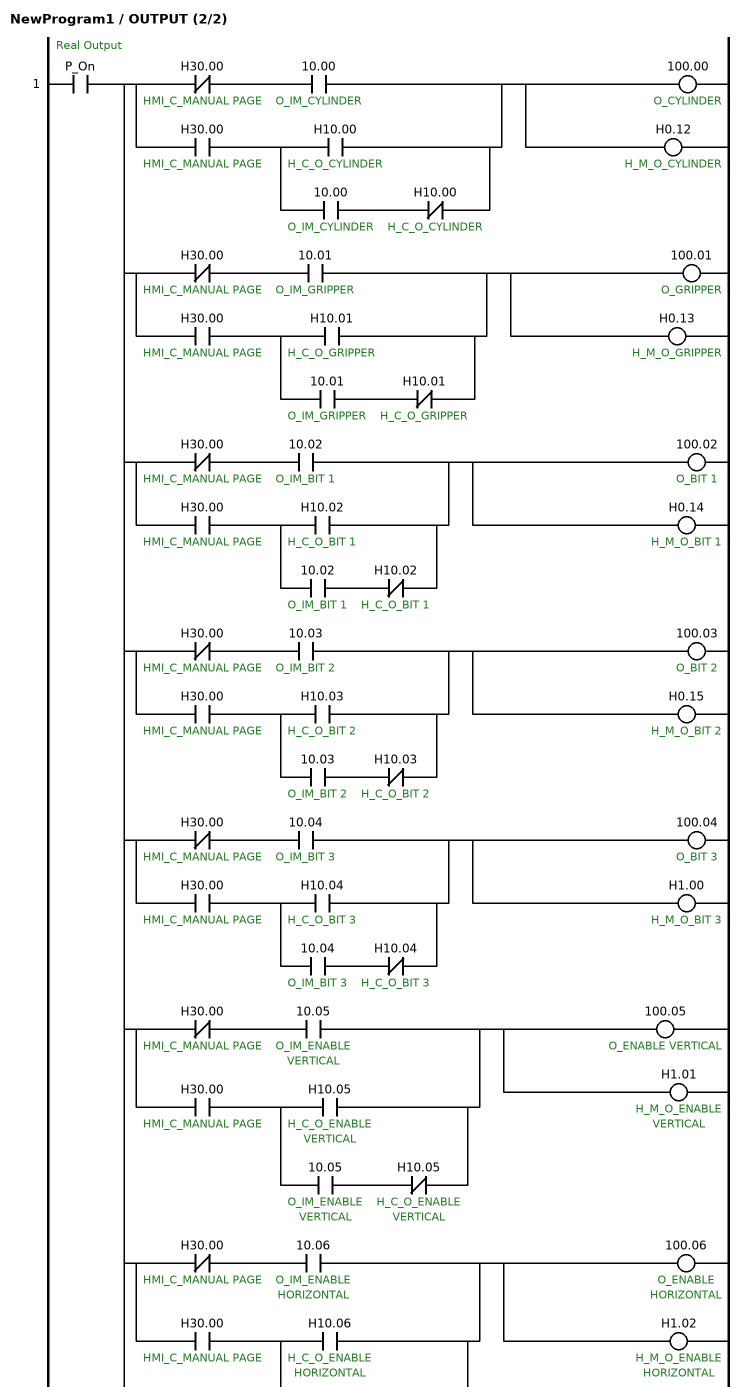
; [picture p48: NewProgram1 / OUTPUT, rungs 1-1]

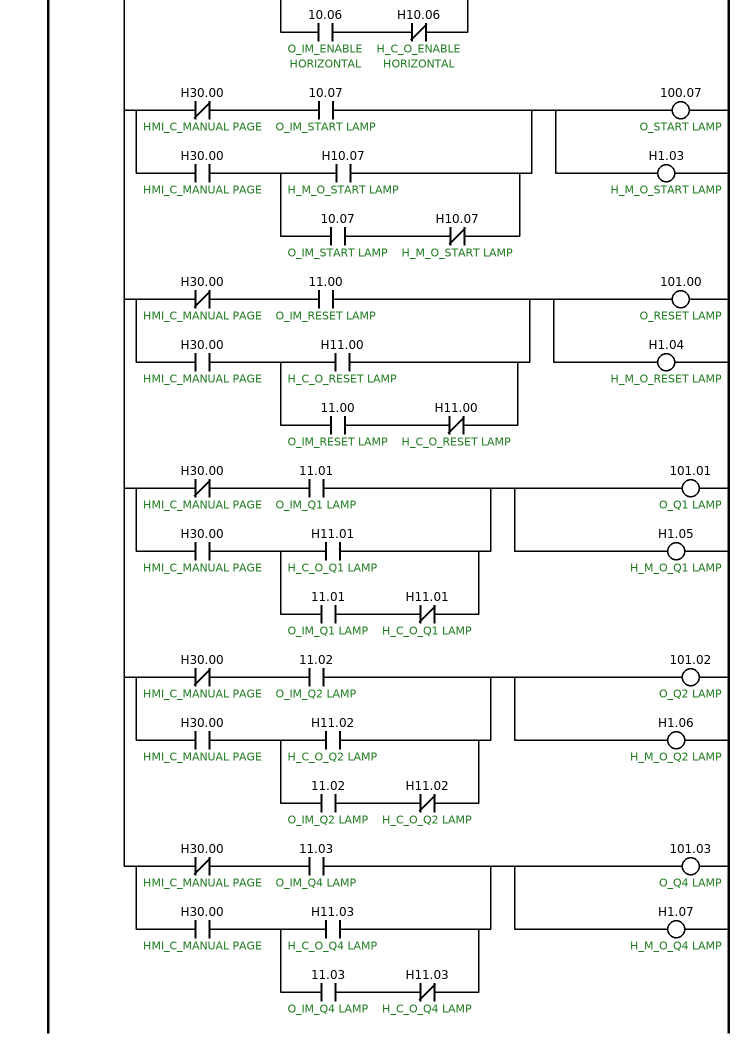
; rung 1: Real Output
LD P_On
OUT TR0
LDNOT H30.00  ; HMI_C_MANUAL PAGE
AND 10.00  ; O_IM_CYLINDER
LD H30.00  ; HMI_C_MANUAL PAGE
LD H10.00  ; H_C_O_CYLINDER
LD 10.00  ; O_IM_CYLINDER
ANDNOT H10.00  ; H_C_O_CYLINDER
ORLD
ANDLD
ORLD
ANDLD
OUT 100.00  ; O_CYLINDER
OUT H0.12  ; H_M_O_CYLINDER
LD TR0
LDNOT H30.00  ; HMI_C_MANUAL PAGE
AND 10.01  ; O_IM_GRIPPER
LD H30.00  ; HMI_C_MANUAL PAGE
LD H10.01  ; H_C_O_GRIPPER
LD 10.01  ; O_IM_GRIPPER
ANDNOT H10.01  ; H_C_O_GRIPPER
ORLD
ANDLD
ORLD
ANDLD
OUT 100.01  ; O_GRIPPER
OUT H0.13  ; H_M_O_GRIPPER
LD TR0
LDNOT H30.00  ; HMI_C_MANUAL PAGE
AND 10.02  ; O_IM_BIT 1
LD H30.00  ; HMI_C_MANUAL PAGE
LD H10.02  ; H_C_O_BIT 1
LD 10.02  ; O_IM_BIT 1
ANDNOT H10.02  ; H_C_O_BIT 1
ORLD
ANDLD
ORLD
ANDLD
OUT 100.02  ; O_BIT 1
OUT H0.14  ; H_M_O_BIT 1
LD TR0
LDNOT H30.00  ; HMI_C_MANUAL PAGE
AND 10.03  ; O_IM_BIT 2
LD H30.00  ; HMI_C_MANUAL PAGE
LD H10.03  ; H_C_O_BIT 2
LD 10.03  ; O_IM_BIT 2
ANDNOT H10.03  ; H_C_O_BIT 2
ORLD
ANDLD
ORLD
ANDLD
OUT 100.03  ; O_BIT 2
OUT H0.15  ; H_M_O_BIT 2
LD TR0
LDNOT H30.00  ; HMI_C_MANUAL PAGE
AND 10.04  ; O_IM_BIT 3
LD H30.00  ; HMI_C_MANUAL PAGE
LD H10.04  ; H_C_O_BIT 3
LD 10.04  ; O_IM_BIT 3
ANDNOT H10.04  ; H_C_O_BIT 3
ORLD
ANDLD
ORLD
ANDLD
OUT 100.04  ; O_BIT 3
OUT H1.00  ; H_M_O_BIT 3
LD TR0
LDNOT H30.00  ; HMI_C_MANUAL PAGE
AND 10.05  ; O_IM_ENABLE VERTICAL
LD H30.00  ; HMI_C_MANUAL PAGE
LD H10.05  ; H_C_O_ENABLE VERTICAL
LD 10.05  ; O_IM_ENABLE VERTICAL
ANDNOT H10.05  ; H_C_O_ENABLE VERTICAL
ORLD
ANDLD
ORLD
ANDLD
OUT 100.05  ; O_ENABLE VERTICAL
OUT H1.01  ; H_M_O_ENABLE VERTICAL
LD TR0
LDNOT H30.00  ; HMI_C_MANUAL PAGE
AND 10.06  ; O_IM_ENABLE HORIZONTAL
LD H30.00  ; HMI_C_MANUAL PAGE
LD H10.06  ; H_C_O_ENABLE HORIZONTAL
LD 10.06  ; O_IM_ENABLE HORIZONTAL
ANDNOT H10.06  ; H_C_O_ENABLE HORIZONTAL
ORLD
ANDLD
ORLD
ANDLD
OUT 100.06  ; O_ENABLE HORIZONTAL
OUT H1.02  ; H_M_O_ENABLE HORIZONTAL
LD TR0
LDNOT H30.00  ; HMI_C_MANUAL PAGE
AND 10.07  ; O_IM_START LAMP
LD H30.00  ; HMI_C_MANUAL PAGE
LD H10.07  ; H_M_O_START LAMP
LD 10.07  ; O_IM_START LAMP
ANDNOT H10.07  ; H_M_O_START LAMP
ORLD
ANDLD
ORLD
ANDLD
OUT 100.07  ; O_START LAMP
OUT H1.03  ; H_M_O_START LAMP
LD TR0
LDNOT H30.00  ; HMI_C_MANUAL PAGE
AND 11.00  ; O_IM_RESET LAMP
LD H30.00  ; HMI_C_MANUAL PAGE
LD H11.00  ; H_C_O_RESET LAMP
LD 11.00  ; O_IM_RESET LAMP
ANDNOT H11.00  ; H_C_O_RESET LAMP
ORLD
ANDLD
ORLD
ANDLD
OUT 101.00  ; O_RESET LAMP
OUT H1.04  ; H_M_O_RESET LAMP
LD TR0
LDNOT H30.00  ; HMI_C_MANUAL PAGE
AND 11.01  ; O_IM_Q1 LAMP
LD H30.00  ; HMI_C_MANUAL PAGE
LD H11.01  ; H_C_O_Q1 LAMP
LD 11.01  ; O_IM_Q1 LAMP
ANDNOT H11.01  ; H_C_O_Q1 LAMP
ORLD
ANDLD
ORLD
ANDLD
OUT 101.01  ; O_Q1 LAMP
OUT H1.05  ; H_M_O_Q1 LAMP
LD TR0
LDNOT H30.00  ; HMI_C_MANUAL PAGE
AND 11.02  ; O_IM_Q2 LAMP
LD H30.00  ; HMI_C_MANUAL PAGE
LD H11.02  ; H_C_O_Q2 LAMP
LD 11.02  ; O_IM_Q2 LAMP
ANDNOT H11.02  ; H_C_O_Q2 LAMP
ORLD
ANDLD
ORLD
ANDLD
OUT 101.02  ; O_Q2 LAMP
OUT H1.06  ; H_M_O_Q2 LAMP
LD TR0
LDNOT H30.00  ; HMI_C_MANUAL PAGE
AND 11.03  ; O_IM_Q4 LAMP
LD H30.00  ; HMI_C_MANUAL PAGE
LD H11.03  ; H_C_O_Q4 LAMP
LD 11.03  ; O_IM_Q4 LAMP
ANDNOT H11.03  ; H_C_O_Q4 LAMP
ORLD
ANDLD
ORLD
ANDLD
OUT 101.03  ; O_Q4 LAMP
OUT H1.07  ; H_M_O_Q4 LAMP

### Section END
; rung 0
END(001)